// TIA Portal V20 export
// export: Created 2025-12-01T14:57:09.7383111Z, ExportSetting None, DisplayName Totally Integrated Automation Portal, DisplayVersion V20 Update 3, DisplayName TIA Portal Openness, DisplayVersion V20 Update 3, DisplayName TIA Portal Version Control Interface, DisplayVersion V20 Update 3, DisplayName STEP 7 Professional, DisplayVersion V20 Update 3, DisplayName STEP 7 Safety, DisplayVersion V20 Update 2, DisplayName WinCC Basic/Comfort/Advanced, DisplayVersion V20 Update 3, DisplayName WinCC Professional, DisplayVersion V20 Update 3, DisplayName WinCC Unified, DisplayVersion V20 Update 3
FUNCTION "FC723_InsertarUT_EnMesa" : Void   // FC723, LAD
TITLE = "InsertarUT_EnMesa" - Creacion de una UT en Mesa
{ S7_Optimized_Access := 'FALSE' }
AUTHOR : TRACKING
NAME : 20130301
VERSION : 3.0
// Mckey 0 - Y al final de la Mesa
// - Buscar una UT Libre
// - Buscar el final de la Mesa
// - Modificar datos de las UT's - Insertar
// stored: AutoNumber false, SetENOAutomatically false
   VAR_INPUT
      MesaActual : UInt;
   END_VAR
   VAR_OUTPUT
      NumeroUT : UInt;
   END_VAR
   VAR_TEMP
      NumUT : UInt;   // Numero UT
      UltimaUT : UInt;
      ValorReturn : Int;
      Cero : Byte;
   END_VAR
BEGIN

NETWORK
TITLE = Inicilizar
////////////////////////////////////////////////////////////////////////
// Inicializa las variables
      L     0;
      T     #NumeroUT;
      T     #NumUT;


///////////////////////////////////////////////////////////////////////////
///////////////////////////////////////////////////////////////////////////
///////////////////////////////////////////////////////////////////////////
/// --- Distribucion Dependiendo del Tipo de JDT (ACTUAL o VIEJO)
      SET;
      A     "Activar_JdTAntiguo";
      JC    Final_Funcion;



NETWORK
TITLE = Buscar una UT Libre
////////////////////////////////////////////////////////////////////////
////////////////////////////////////////////////////////////////////////
////////////////////////////////////////////////////////////////////////
      L     1;
      T     #NumUT;

Bucle_BuquedaUT:NOP   0;
      L     "DB812_UTs_Control".UT[#NumUT].MesaActual;
      L     0;  // Esta Vacia - 0
      ==I;
      JC    Encontrada_NuevaUT;

      L     #NumUT;  // A la siguiente UT
      L     1;
      +I;
      T     #NumUT;

      L     #NumUT;
      L     "CTE_MaxUTs";  // Si hemos llegado a la Ultima UT
      <=I;
      JC    Bucle_BuquedaUT;

      L     0;
      T     #NumUT;
      JU    Final_Funcion;



NETWORK
TITLE = UT EnContrada
////////////////////////////////////////////////////////////////////////
////////////////////////////////////////////////////////////////////////
////////////////////////////////////////////////////////////////////////
// Ya tenemos la UT nueva, Y es la unica.
// Rellanar campos de la base de datos con lo basico

Encontrada_NuevaUT:NOP   0;

////////////////////////////////////////////////////////////////////////////////
// Limpieza de la UT

      L     0;  // Valor a rellenar
      T     #Cero;

// Borrado del DB de Control de la UT
      CALL  FILL
      ( BVAL    := #Cero,
        RET_VAL := #ValorReturn,
        BLK     := "DB812_UTs_Control".UT[#NumeroUT]
      );

// Borrado del DB de la Rutas de la UT
      CALL  FILL
      ( BVAL    := #Cero,
        RET_VAL := #ValorReturn,
        BLK     := "DB813_UTs_Ruta".UT[#NumeroUT]
      );

// Borrado del DB de los Datos de la UT
      CALL  FILL
      ( BVAL    := #Cero,
        RET_VAL := #ValorReturn,
        BLK     := "DB814_UTs_Etiqueta".UT[#NumeroUT]
      );
      CALL  FILL
      ( BVAL    := #Cero,
        RET_VAL := #ValorReturn,
        BLK     := "DB815_UTs_Datos".UT[#NumeroUT]
      );
      CALL  FILL
      ( BVAL    := #Cero,
        RET_VAL := #ValorReturn,
        BLK     := "DB816_UTs_TextoPantalla".UT[#NumeroUT]
      );
      CALL  FILL
      ( BVAL    := #Cero,
        RET_VAL := #ValorReturn,
        BLK     := "DB820_UTs_DatosQUBIQA".UT[#NumeroUT]
      );
      CALL  FILL
      ( BVAL    := #Cero,
        RET_VAL := #ValorReturn,
        BLK     := "DB821_UTs_DatosIKPAL".UT[#NumeroUT]
      );


////////////////////////////////////////////////////////////////////////////////
// Relleno datos Basicos de la UT
      L     #MesaActual;  // Poner la mesa correcta
      L     "CTE_OffsetMesa";  // +Offet
      +I;
      T     "DB812_UTs_Control".UT[#NumUT].MesaActual;



NETWORK
TITLE = Colar la UT en el final de la Cola de Mesa -- Previo
////////////////////////////////////////////////////////////////////////
////////////////////////////////////////////////////////////////////////
////////////////////////////////////////////////////////////////////////
// Empiezo a recorrer los datos de UT en la Mesa
// Miro primero si hay alguna UT en la Mesa
      L     "DB810_ColasMesas".Colas[#MesaActual].UT_PrimeraMesa;
      T     #UltimaUT;

      L     #UltimaUT;
      L     0;
      <>I;  // Hay UT's en la Mesa
      JC    HayUT_EnColaMesa;
      JU    NoHayUT_EnColaMesa;



NETWORK
TITLE = No Hay UTs en la Cola de la Mesa
////////////////////////////////////////////////////////////////////////
////////////////////////////////////////////////////////////////////////
////////////////////////////////////////////////////////////////////////
// No hay ninguna, solo hay que poner cual es la primera de la mesa
NoHayUT_EnColaMesa:NOP   0;
      L     #NumUT;
      T     "DB810_ColasMesas".Colas[#MesaActual].UT_PrimeraMesa;

      JU    Final_Funcion;



NETWORK
TITLE = Hay UTs en la Cola de la Mesa
////////////////////////////////////////////////////////////////////////
////////////////////////////////////////////////////////////////////////
////////////////////////////////////////////////////////////////////////
// Si hay UT's en la mesa, hay que buscar la ultima
HayUT_EnColaMesa:NOP   0;
      L     "DB812_UTs_Control".UT[#UltimaUT].UT_SiguienteMesa;
      L     0;  // Es la Ultima
      ==I;
      JC    EncontradaUltimaUT_EnColaMesa;

      L     "DB812_UTs_Control".UT[#UltimaUT].UT_SiguienteMesa;
      T     #UltimaUT;

      JU    HayUT_EnColaMesa;


////////////////////////////////////////////////////////////////////////
// Modifico al ultima UT de la Mesa
EncontradaUltimaUT_EnColaMesa:NOP   0;
      L     #NumUT;
      T     "DB812_UTs_Control".UT[#UltimaUT].UT_SiguienteMesa;


////////////////////////////////////////////////////////////////////////
// Moodifico la nueva UT de la Mesa - Nueva Ultima

      L     #UltimaUT;
      T     "DB812_UTs_Control".UT[#NumUT].UT_AnteriorMesa;



NETWORK
TITLE = Final de la funcion
////////////////////////////////////////////////////////////////////////
////////////////////////////////////////////////////////////////////////
////////////////////////////////////////////////////////////////////////
Final_Funcion:NOP   0;

// Devolucion de la UT
      L     #NumUT;
      T     #NumeroUT;



END_FUNCTION
